// TIA Portal V18 export
// export: Created 2025-12-01T17:53:06.9243284Z, ExportSetting None, DisplayName Totally Integrated Automation Portal, DisplayVersion V18 Update 5, DisplayName TIA Portal Openness, DisplayVersion V18 Update 5, DisplayName TIA Portal Teamcenter Gateway, DisplayVersion V18, DisplayName TIA Portal Version Control Interface, DisplayVersion V18, DisplayName STEP 7 Professional, DisplayVersion V18 Update 5, DisplayName STEP 7 Safety, DisplayVersion V18, DisplayName WinCC Professional, DisplayVersion V18 Update 5
Screen "294_Motor_L2"  1280x800, Number=294, Template=02ManualUnit1
  ScreenLayer "Layer_0"
    Button "btnMenu5" at 512,725 size 128x75  TextOff="L-电机2 / L-Motor2", TextOn="L-电机2 / L-Motor2"
      on Click: ActivateScreen(Screen name := , Object number := 0)
    FaceplateInstance "Motor_1" at 70,138 size 273x159  FaceplateTypeName=03 FunctionBlocks@$@202 Conveyer_Line@$@202.2 HMI@$@Motor V 0.0.7
      MotorControl := MotorControl_Dev{4}
      InterfacePropertyText "TextName"  Text="L_下料电机 / L_Unloading Motor"
    FaceplateInstance "Motor_2" at 370,138 size 316x159  FaceplateTypeName=03 FunctionBlocks@$@202 Conveyer_Line@$@202.2 HMI@$@Motor V 0.0.7
      MotorControl := MotorControl_Dev{17}
      InterfacePropertyText "TextName"  Text="L_空托盘上料电机 / L_EmptyPalletLoadingMotor / H流线电机"
    Button "按钮_9" at 128,725 size 128x75  PictureOff=向右箭头_0, TextOff="L-气缸1 / L-Cylinder1", TextOn="L-气缸1 / L-Cylinder1"
      on Click: ActivateScreen(Screen name := 290_Cylinder_L1, Object number := 0)
    Button "btnMenu6" at 640,725 size 128x75  StyleItem=BtnNormal20
    Button "btnMenu6_1" at 768,725 size 128x75  StyleItem=BtnNormal20
    Button "btnMenu4" at 384,725 size 128x75  TextOff="L-气缸2 / L-Cylinder2", TextOn="L-气缸2 / L-Cylinder2"
      on Click: ActivateScreen(Screen name := 293_Cylinder_L2, Object number := 0)
    Button "btnMenu7" at 896,725 size 128x75
    Button "btnMenu7_1" at 1024,725 size 128x75
    Button "btnMenu4_1" at 256,725 size 128x75  TextOff="L-电机1 / L-Motor1", TextOn="L-电机1 / L-Motor1"
      on Click: ActivateScreen(Screen name := 291_Motor_L1, Object number := 0)
